FUNCTION_BLOCK XtsPart EXTENDS CyclicBase
VAR
	_MyInterface : Tc3_XTS_Utility.I_TcIoXtsXpuPart;
	XtsIoEnvInitialiseState : INT;
	MyModuleCount : UDINT;
	PartDriveState: Tc3_XTS_Utility.DriveState;
	_ReadyToEnable: BOOL;
	MyModules : ARRAY[0..TcIoXtsEnvironmentParameterList.MaxModulesPerPart] OF XtsMotorModule;
	ModuleIndex: UDINT := 1;
	CurrentErrorId : UDINT;
	InSim : BOOL;
	PartName: STRING;
	IsDCLinkReady: BOOL;
END_VAR

METHOD PUBLIC  Cycle : HRESULT
VAR
	i : INT;
	tempErrorID : UDINT;
END_VAR
PartDriveState := _MyInterface.GetDriveState();
IsDCLinkReady := _MyInterface.GetIsDcLinkVoltageReady();
IF HasError() THEN
	FOR i := 0 TO (UDINT_TO_UINT(MyModuleCount) - 1) DO
		tempErrorID := MyModules[i].GetLatestDiagMessage();
		IF tempErrorID > CurrentErrorId THEN
			CurrentErrorId := tempErrorID;
		END_IF
	END_FOR
END_IF
FOR i := 0 TO (UDINT_TO_UINT(MyModuleCount) - 1) DO
	MyModules[i].Cycle();
END_FOR
END_METHOD

METHOD GetCurrentError : UDINT
VAR_INPUT
END_VAR
GetCurrentError := CurrentErrorId;
END_METHOD

METHOD HasError : BOOL
VAR_INPUT
END_VAR
HasError := PartDriveState = DriveState.Fault OR PartDriveState = DriveState.FaultReactionActive OR NOT _MyInterface.GetIsDcLinkVoltageReady();
END_METHOD

METHOD Initialise : HRESULT
VAR
	i : INT;
END_VAR
Initialise := -1;
CASE XtsIoEnvInitialiseState OF
	0:
		IF _MyInterface <> 0 THEN
			XtsIoEnvInitialiseState := 1;
		ELSE
			XtsIoEnvInitialiseState := 999;
		END_IF
	1:
		MyModuleCount := _MyInterface.GetModuleCount();
		IF InSim THEN
			XtsIoEnvInitialiseState := 3;
			FOR i := 0 TO UDINT_TO_UINT(MyModuleCount - 1) DO
				MyModules[i].SetInSim();
			END_FOR
			InSim := true;
		ELSE
			FOR i := 0 TO UDINT_TO_UINT(MyModuleCount - 1) DO
				MyModules[i].MyModuleInterface := _MyInterface.ModuleTcIo(i + 1);
			END_FOR
			XtsIoEnvInitialiseState := 2;
		END_IF
		
	2:
		XtsIoEnvInitialiseState := 3;
		FOR i := 0 TO UDINT_TO_UINT(MyModuleCount-1) DO
			IF MyModules[i].Initialise() <> 2 THEN
				XtsIoEnvInitialiseState := 2;
			END_IF
		END_FOR
	3:
		PartName := _MyInterface.P_ObjectName;
		Initialise := 0;
END_CASE
END_METHOD

METHOD Is24VBusOK : BOOL
VAR
	i : INT;
END_VAR
Is24VBusOK := TRUE;
FOR i := 0 TO (UDINT_TO_UINT(MyModuleCount) - 1) DO
	IF MyModules[i].Is24VOK() = -1 THEN
		Is24VBusOK := FALSE;
	END_IF
END_FOR
END_METHOD

METHOD Is48VBusOK : BOOL
VAR
	i : INT;
END_VAR
Is48VBusOK := TRUE;
FOR i := 0 TO (UDINT_TO_UINT(MyModuleCount) - 1) DO
	IF MyModules[i].Is48VOK() = -1 THEN
		Is48VBusOK := FALSE;
	END_IF
END_FOR
END_METHOD

PROPERTY MyXtsIoEnvInterface : I_TcIoXtsXpuPart
GET
MyXtsIoEnvInterface := _MyInterface;
END_GET
SET
_MyInterface := MyXtsIoEnvInterface;
END_SET
END_PROPERTY

METHOD ResetNct : BOOL
VAR_INPUT
END_VAR
ResetNct := _MyInterface.TriggerNctReset();
END_METHOD

METHOD ResetPart : BOOL
VAR
	i : INT;
END_VAR
ResetPart := _MyInterface.TriggerReset();
IF NOT InSim THEN
	FOR i := 0 TO (UDINT_TO_UINT(MyModuleCount) - 1) DO
		MyModules[i].AckDiagMsgs();
	END_FOR
END_IF	
CurrentErrorId := 0;
END_METHOD

METHOD SetInSim : HRESULT
VAR_INPUT
END_VAR
InSim := true;
END_METHOD

METHOD SetPartOriginTransform : BOOL
VAR_INPUT
	OriginTransform: Tc3_XTS_Utility.ST_OriginTransform;
END_VAR
_MyInterface.SetOriginTransform(OriginTransform);
END_METHOD

END_FUNCTION_BLOCK

(* stored: Version 1.1.0.1
   POU XtsPart: Id {39541d00-22ec-4750-829d-4864a624597e}, SpecialFunc None
   Method Cycle: Id {6aa26807-846b-4168-ab87-fb4c66b138eb}
   Method GetCurrentError: Id {397b05da-5d11-4ea0-a858-00e1feeb8a6c}
   Method HasError: Id {1ff560a3-4b5c-4bd0-a848-6c6a900a7eef}
   Method Initialise: Id {f7bcb601-a320-4f3f-bcf3-5ec4e45a7245}
   Method Is24VBusOK: Id {d79d6eda-1f90-4384-9dda-ac7f4aaa7f07}
   Method Is48VBusOK: Id {44113d88-367f-494b-87cf-4655fd94d258}
   Property MyXtsIoEnvInterface: Id {b5f6c838-c909-4a11-9656-9e449699aee4}
   Get Get: Id {249dae7e-fa2b-4c2d-a421-a33d92e9b50d}
   Set Set: Id {436f8d77-48c4-4edc-81e4-5821f3038a93}
   Method ResetNct: Id {ada2aac2-9e86-42a2-81c2-fb2391256788}
   Method ResetPart: Id {a2c1bf74-a00f-4e37-abd0-e53201644a52}
   Method SetInSim: Id {273102d0-bbf8-41a5-af45-2632119808d5}
   Method SetPartOriginTransform: Id {8b2a2802-8f42-46b7-9bd8-2e1c722c9321} *)
